// TIA Portal V15.1 export
// export: Created 2024-06-21T08:41:04.5665723Z, ExportSetting WithDefaults, DisplayName Totally Integrated Automation Portal, DisplayVersion V15.1 Update 5, DisplayName TIA Portal Openness, DisplayVersion V15.1 Update 5, DisplayName SINAMICS Startdrive Advanced, DisplayVersion V15.1, DisplayName G130, G150, S120, S150, SINAMICS MV, S210, DisplayVersion V15.1, DisplayName G110M, G120, G120C, G120D, G120P, DisplayVersion V15.1, DisplayName STEP 7 Professional, DisplayVersion V15.1 Update 5, DisplayName STEP 7 Safety, DisplayVersion V15.1, DisplayName WinCC Professional, DisplayVersion V15.1 Update 5, DisplayName SIMATIC Visualization Architect, DisplayVersion V15.1
FUNCTION_BLOCK "LProcVlvPidFbk"   // FB1734, FBD
TITLE = LProcVlvPidFbk
{ S7_Optimized_Access := 'FALSE' }
AUTHOR : VCC
FAMILY : ProcEq
NAME : PIDDONFb
VERSION : 0.1
// ================================================================================
// This is a Valve/Damper PID-controller module.
// The module contains: 
// 1 analog input function block
// a PID controller loop and a DO controller to activate the contactors Open
// and Close
// There is a feedback of position of the valve.
// ================================================================================
// stored: AutoNumber false, IsIECCheckEnabled false, SetENOAutomatically False, UDAEnableTagReadback false
   VAR_INPUT
      I_ExtSP1_Value { ExternalAccessible := 'False'; ExternalVisible := 'False'; ExternalWritable := 'False'} : Real;   // External Set-point 1
      I_ForcedValue { ExternalAccessible := 'False'; ExternalVisible := 'False'; ExternalWritable := 'False'} : Real;   // Pid Output Forced value (when I_ForceOutput is true)
      I_DO_POS { ExternalAccessible := 'False'; ExternalVisible := 'False'; ExternalWritable := 'False'} : Int;   // Feedback position DO controller
      I_DetSetLimit { ExternalAccessible := 'False'; ExternalVisible := 'False'; ExternalWritable := 'False'} : Real;   // Detection Set Limit
      I_DetResetLimit { ExternalAccessible := 'False'; ExternalVisible := 'False'; ExternalWritable := 'False'} : Real := 100.0;   // Detection Reset Limit
      I_PV_AnInput { ExternalAccessible := 'False'; ExternalVisible := 'False'; ExternalWritable := 'False'} : Int;   // Process Value Analog Input
      I_SPReq : Int;   // Index Set-point Request
      I_MaxTime { ExternalAccessible := 'False'; ExternalVisible := 'False'; ExternalWritable := 'False'} : DInt;   // Maximum Time to get Set and reset detections
      I_ExtSP1 { ExternalAccessible := 'False'; ExternalVisible := 'False'; ExternalWritable := 'False'} : Bool;   // External Set-point 1 Request
      I_ControllerON { ExternalAccessible := 'False'; ExternalVisible := 'False'; ExternalWritable := 'False'} : Bool;   // Start Pid Controller
      I_ForceOutput : Bool;   // Force Pid Output Value to Forced Value
      I_DetSet { ExternalAccessible := 'False'; ExternalVisible := 'False'; ExternalWritable := 'False'} : Bool;   // Detection Set
      I_DetReset { ExternalAccessible := 'False'; ExternalVisible := 'False'; ExternalWritable := 'False'} : Bool;   // Detection Reset
      I_AutoSetReq { ExternalAccessible := 'False'; ExternalVisible := 'False'; ExternalWritable := 'False'} : Bool;   // Set Valve/Damper from sequence or equation
      I_AutoResetReq { ExternalAccessible := 'False'; ExternalVisible := 'False'; ExternalWritable := 'False'} : Bool;   // Reset Valve/Damper from sequence or equation
      I_InterlockSetOk { ExternalAccessible := 'False'; ExternalVisible := 'False'; ExternalWritable := 'False'} : Bool;   // Interlock Set Direction
      I_InterlockResetOk { ExternalAccessible := 'False'; ExternalVisible := 'False'; ExternalWritable := 'False'} : Bool;   // Interlock Reset Direction
      I_EnableAlarm { ExternalAccessible := 'False'; ExternalVisible := 'False'; ExternalWritable := 'False'} : Bool;   // Enable Alarms
      I_PBSetPBResetAllAutoSel { ExternalAccessible := 'False'; ExternalVisible := 'False'; ExternalWritable := 'False'} : Struct   // Set PB activated - Reset PB activated - All HMI Auto selected
         HMI1SetPB { ExternalAccessible := 'False'; ExternalVisible := 'False'; ExternalWritable := 'False'} : Bool;   // Set PB activated on HMI1
         HMI1ResetPB { ExternalAccessible := 'False'; ExternalVisible := 'False'; ExternalWritable := 'False'} : Bool;   // Reset PB activated on HMI1
         HMI1AllHMIAutoSel { ExternalAccessible := 'False'; ExternalVisible := 'False'; ExternalWritable := 'False'} : Bool;   // All HMI Auto selected on HMI1
         HMI2SetPB { ExternalAccessible := 'False'; ExternalVisible := 'False'; ExternalWritable := 'False'} : Bool;   // Set PB activated on HMI2
         HMI2ResetPB { ExternalAccessible := 'False'; ExternalVisible := 'False'; ExternalWritable := 'False'} : Bool;   // Reset PB activated on HMI2
         HMI2AllHMIAutoSel { ExternalAccessible := 'False'; ExternalVisible := 'False'; ExternalWritable := 'False'} : Bool;   // All HMI Auto selected on HMI2
         HMI3SetPB { ExternalAccessible := 'False'; ExternalVisible := 'False'; ExternalWritable := 'False'} : Bool;   // Set PB activated on HMI3
         HMI3ResetPB { ExternalAccessible := 'False'; ExternalVisible := 'False'; ExternalWritable := 'False'} : Bool;   // Reset PB activated on HMI3
         HMI3AllHMIAutoSel { ExternalAccessible := 'False'; ExternalVisible := 'False'; ExternalWritable := 'False'} : Bool;   // All HMI Auto selected on HMI3
         HMI4SetPB { ExternalAccessible := 'False'; ExternalVisible := 'False'; ExternalWritable := 'False'} : Bool;   // Set PB activated on HMI4
         HMI4ResetPB { ExternalAccessible := 'False'; ExternalVisible := 'False'; ExternalWritable := 'False'} : Bool;   // Reset PB activated on HMI4
         HMI4AllHMIAutoSel { ExternalAccessible := 'False'; ExternalVisible := 'False'; ExternalWritable := 'False'} : Bool;   // All HMI Auto selected on HMI4
         HMI5SetPB { ExternalAccessible := 'False'; ExternalVisible := 'False'; ExternalWritable := 'False'} : Bool;   // Set PB activated on HMI5
         HMI5ResetPB { ExternalAccessible := 'False'; ExternalVisible := 'False'; ExternalWritable := 'False'} : Bool;   // Reset PB activated on HMI5
         HMI5AllHMIAutoSel { ExternalAccessible := 'False'; ExternalVisible := 'False'; ExternalWritable := 'False'} : Bool;   // All HMI Auto selected on HMI5
         StartPBSel { ExternalAccessible := 'False'; ExternalVisible := 'False'; ExternalWritable := 'False'} : Bool;   // Start is activated
         AlarmResetPBSel { ExternalAccessible := 'False'; ExternalVisible := 'False'; ExternalWritable := 'False'} : Bool;   // Alarm reset is activated
      END_STRUCT;
      I_UpperLevelAlarmA { ExternalAccessible := 'False'; ExternalVisible := 'False'; ExternalWritable := 'False'} : Bool;   // Alarm A from Upper Level
      I_UpperLevelAlarmB { ExternalAccessible := 'False'; ExternalVisible := 'False'; ExternalWritable := 'False'} : Bool;   // Alarm B from Upper Level
      I_EnHHHAlarm { ExternalAccessible := 'False'; ExternalVisible := 'False'; ExternalWritable := 'False'} : Bool;   // Enable HHH Limit Alarm
      I_ResHHHAlarm { ExternalAccessible := 'False'; ExternalVisible := 'False'; ExternalWritable := 'False'} : Bool;   // Reset HHH Limit Alarm
      I_EnHHAlarm { ExternalAccessible := 'False'; ExternalVisible := 'False'; ExternalWritable := 'False'} : Bool;   // Enable HH Limit Alarm
      I_ResHHAlarm { ExternalAccessible := 'False'; ExternalVisible := 'False'; ExternalWritable := 'False'} : Bool;   // Reset HH Limit Alarm
      I_EnHAlarm { ExternalAccessible := 'False'; ExternalVisible := 'False'; ExternalWritable := 'False'} : Bool;   // Enable H Limit Alarm
      I_ResHAlarm { ExternalAccessible := 'False'; ExternalVisible := 'False'; ExternalWritable := 'False'} : Bool;   // Reset H Limit Alarm
      I_EnLAlarm { ExternalAccessible := 'False'; ExternalVisible := 'False'; ExternalWritable := 'False'} : Bool;   // Enable L Limit Alarm
      I_ResLAlarm { ExternalAccessible := 'False'; ExternalVisible := 'False'; ExternalWritable := 'False'} : Bool;   // Reset L Limit Alarm
      I_EnLLAlarm { ExternalAccessible := 'False'; ExternalVisible := 'False'; ExternalWritable := 'False'} : Bool;   // Enable LL Limit Alarm
      I_ResLLAlarm { ExternalAccessible := 'False'; ExternalVisible := 'False'; ExternalWritable := 'False'} : Bool;   // Reset LL Limit Alarm
      I_EnLLLAlarm { ExternalAccessible := 'False'; ExternalVisible := 'False'; ExternalWritable := 'False'} : Bool;   // Enable LLL Limit Alarm
      I_ResLLLAlarm { ExternalAccessible := 'False'; ExternalVisible := 'False'; ExternalWritable := 'False'} : Bool;   // Reset LLL Limit Alarm
      C_ManualForcedUsed { ExternalAccessible := 'False'; ExternalVisible := 'False'; ExternalWritable := 'False'} : Bool;   // Manual Forced is used (=true)
      C_DetSetUsed { ExternalAccessible := 'False'; ExternalVisible := 'False'; ExternalWritable := 'False'} : Bool;   // Detection Set used (true=used)
      C_DetResetUsed { ExternalAccessible := 'False'; ExternalVisible := 'False'; ExternalWritable := 'False'} : Bool;   // Detection Reset used (true=used)
   END_VAR
   VAR_OUTPUT
      O_PV : Real;   // Process Value scaled
      O_SP : Real;   // Setpoint used in controller
      O_PosFbk : Real;   // Damp/Valve position feedback value used in controller
      O_LMN : Real;   // Pid Output value
      O_SetFbk : Bool;   // Valve/Damper in Set position
      O_ResetFbk : Bool;   // Valve/Damper in Reset position
      O_SetCmd { ExternalAccessible := 'False'; ExternalVisible := 'False'; ExternalWritable := 'False'} : Bool;   // Valve/Damper Set command
      O_ResetCmd { ExternalAccessible := 'False'; ExternalVisible := 'False'; ExternalWritable := 'False'} : Bool;   // Valve/Damper Reset command
      O_AlarmABCondition { ExternalAccessible := 'False'; ExternalVisible := 'False'; ExternalWritable := 'False'} : Bool;   // Alarm AB condition
      O_AlarmA { ExternalAccessible := 'False'; ExternalVisible := 'False'; ExternalWritable := 'False'} : Bool;   // Summation Alarm A
      O_AlarmB { ExternalAccessible := 'False'; ExternalVisible := 'False'; ExternalWritable := 'False'} : Bool;   // Summation Alarm B
      O_AlarmC { ExternalAccessible := 'False'; ExternalVisible := 'False'; ExternalWritable := 'False'} : Bool;   // Summation Alarm C
      O_AlarmD { ExternalAccessible := 'False'; ExternalVisible := 'False'; ExternalWritable := 'False'} : Bool;   // Summation Alarm D
      O_HHHAlarm { ExternalAccessible := 'False'; ExternalVisible := 'False'; ExternalWritable := 'False'} : Bool;   // HHH Alarm
      O_HHAlarm { ExternalAccessible := 'False'; ExternalVisible := 'False'; ExternalWritable := 'False'} : Bool;   // HH Alarm
      O_HAlarm { ExternalAccessible := 'False'; ExternalVisible := 'False'; ExternalWritable := 'False'} : Bool;   // H Alarm
      O_LAlarm { ExternalAccessible := 'False'; ExternalVisible := 'False'; ExternalWritable := 'False'} : Bool;   // L Alarm
      O_LLAlarm { ExternalAccessible := 'False'; ExternalVisible := 'False'; ExternalWritable := 'False'} : Bool;   // LL Alarm
      O_LLLAlarm { ExternalAccessible := 'False'; ExternalVisible := 'False'; ExternalWritable := 'False'} : Bool;   // LLL Alarm
      O_HHHReached { ExternalAccessible := 'False'; ExternalVisible := 'False'; ExternalWritable := 'False'} : Bool;   // High High High Limit Reached
      O_HHReached { ExternalAccessible := 'False'; ExternalVisible := 'False'; ExternalWritable := 'False'} : Bool;   // High High Limit Reached
      O_HReached { ExternalAccessible := 'False'; ExternalVisible := 'False'; ExternalWritable := 'False'} : Bool;   // High Limit Reached
      O_LReached { ExternalAccessible := 'False'; ExternalVisible := 'False'; ExternalWritable := 'False'} : Bool;   // Low Limit Reached
      O_LLReached { ExternalAccessible := 'False'; ExternalVisible := 'False'; ExternalWritable := 'False'} : Bool;   // Low Low Limit Reached
      O_LLLReached { ExternalAccessible := 'False'; ExternalVisible := 'False'; ExternalWritable := 'False'} : Bool;   // Low Low Low Limit Reached
      H_IAnim { ExternalAccessible := 'False'; ExternalVisible := 'False'; ExternalWritable := 'False'} : Word;   // HMI Animation color of the icon
      H_AlarmWord { ExternalAccessible := 'False'; ExternalVisible := 'False'; ExternalWritable := 'False'} : DWord;   // Alarm Word
   END_VAR
   VAR_IN_OUT
      PV_AnScale : "LProcAnInput6Lim";   // DB for the analogue scaling of Process Value
   END_VAR
   VAR DB_SPECIFIC
      AB_OvTimeAutoSel { ExternalAccessible := 'False'; ExternalVisible := 'False'; ExternalWritable := 'False'} : Bool;   // Alarm Overtime Auto selected
      AD_AcofDetSet { ExternalAccessible := 'False'; ExternalVisible := 'False'; ExternalWritable := 'False'} : Bool;   // Acof Fault Set detection
      AD_AcofDetReset { ExternalAccessible := 'False'; ExternalVisible := 'False'; ExternalWritable := 'False'} : Bool;   // Acof Fault Reset detection
      AD_PV_SensorAlm { ExternalAccessible := 'False'; ExternalVisible := 'False'; ExternalWritable := 'False'} : Bool;   // Process Value sensor alarm
      AD_InterlockSetAlm { ExternalAccessible := 'False'; ExternalVisible := 'False'; ExternalWritable := 'False'} : Bool;   // Interlock Set Alarm
      AD_InterlockResetAlm { ExternalAccessible := 'False'; ExternalVisible := 'False'; ExternalWritable := 'False'} : Bool;   // Interlock Reset Alarm
      H_HMIModeCmd : Word;   // Mode commands from HMI
      H_ActiveHMI : Int;   // Active HMI
      H_NameActiveHMI : String[25];   // Name of the Active HMI
      H_In : Struct   // HMI
         SP2 : Real;   // Set-point 2
         SP3 : Real;   // Set-point 3
         SP4 : Real;   // Set-point 4
         SP5 : Real;   // Set-point 5
         GAIN : Real;   // Pid Proportional Gain
         PID_DEADB_W : Real;   // Pid Deadband width
         LMN_HLM : Real;   // Pid Manipulated value high limit
         LMN_LLM : Real;   // Pid Manipulated value low limit
         TI : Time;   // Pid Reset time
         TD : Time;   // Pid Derivative time
         PULSE_TM : Time;   // Minimum Pulse Time
         BREAK_TM : Time;   // Minimum Break Time
         MTR_TM : Time;   // Motor manipulated time value
         DO_DEADB_W : Real;   // Motor Deadband width
         DO_POS_FAC : Real;   // Factor for feedback of position
         Direct : Bool;   // Pid in Direct mode (output increase if SP>PV)
         P_SEL : Bool;   // Pid P selected
         I_SEL : Bool;   // Pid I selected
         D_SEL : Bool;   // Pid D selected
      END_STRUCT;
      H_Out : Struct   // HMI
         AnInputIAnim : Word;   // HMI Animation color of the icon
         DetSetIAnim : Word;   // HMI Animation color of object
         DetResetIAnim : Word;   // HMI Animation color of object
         ContactorSetIAnim : Word;   // HMI Animation color of object
         ContactorResetIAnim : Word;   // HMI Animation color of object
         Anim : Word;   // HMI Animation of the object
         Anim2 : Word;   // HMI Animation of the object
         Anim3 : Bool;   // HMI Animation bool
         DBnr : Int;   // HMI Animation DB number
      END_STRUCT;
      H_InOut : Struct   // HMI
         Manual_Value : Real;   // Position Setpoint in Manual
         SP1 : Real;   // Set-point 1
      END_STRUCT;
      CYCLE { ExternalAccessible := 'False'; ExternalVisible := 'False'; ExternalWritable := 'False'} : Time := T#100MS;   // Sample time for controller
      PV_AIScaled { ExternalAccessible := 'False'; ExternalVisible := 'False'; ExternalWritable := 'False'} : Real;   // Proces Value: Analog Input after scaling
      PV_PID { ExternalAccessible := 'False'; ExternalVisible := 'False'; ExternalWritable := 'False'} : Real;   // Pid Process value
      SPSel { ExternalAccessible := 'False'; ExternalVisible := 'False'; ExternalWritable := 'False'} : Real;   // Set-point selected
      SP { ExternalAccessible := 'False'; ExternalVisible := 'False'; ExternalWritable := 'False'} : Real;   // Set-point used for Pid regulation
      PosFbk { ExternalAccessible := 'False'; ExternalVisible := 'False'; ExternalWritable := 'False'} : Real;   // Position Feedback (calculation) of the Valve/Damper
      DeadPosOpen { ExternalAccessible := 'False'; ExternalVisible := 'False'; ExternalWritable := 'False'} : Real;   // Calculation Position Open - deadband
      DeadPosClosed { ExternalAccessible := 'False'; ExternalVisible := 'False'; ExternalWritable := 'False'} : Real;   // Calculation Position Closed + deadband
      LMN { ExternalAccessible := 'False'; ExternalVisible := 'False'; ExternalWritable := 'False'} : Real;   // Pid Output value
      DetSet { ExternalAccessible := 'False'; ExternalVisible := 'False'; ExternalWritable := 'False'} : Bool;   // Detection Set
      DetReset { ExternalAccessible := 'False'; ExternalVisible := 'False'; ExternalWritable := 'False'} : Bool;   // Detection Reset
      AutoMode { ExternalAccessible := 'False'; ExternalVisible := 'False'; ExternalWritable := 'False'} : Bool;   // Auto mode
      ManualMode { ExternalAccessible := 'False'; ExternalVisible := 'False'; ExternalWritable := 'False'} : Bool;   // Manual mode
      AutoModeSel { ExternalAccessible := 'False'; ExternalVisible := 'False'; ExternalWritable := 'False'} : Bool;   // Auto Mode Selection from HMI
      ManualModeSel { ExternalAccessible := 'False'; ExternalVisible := 'False'; ExternalWritable := 'False'} : Bool;   // Manual Mode Selection from HMI
      ForcedMan { ExternalAccessible := 'False'; ExternalVisible := 'False'; ExternalWritable := 'False'} : Bool;   // Forced manual active
      AllHMIAutoSel { ExternalAccessible := 'False'; ExternalVisible := 'False'; ExternalWritable := 'False'} : Bool;   // All HMI Auto selected
      Set { ExternalAccessible := 'False'; ExternalVisible := 'False'; ExternalWritable := 'False'} : Bool;   // Controller output Set
      Reset { ExternalAccessible := 'False'; ExternalVisible := 'False'; ExternalWritable := 'False'} : Bool;   // Controller output Reset
      OvTimeAutoSelCond { ExternalAccessible := 'False'; ExternalVisible := 'False'; ExternalWritable := 'False'} : Bool;   // Overtime Auto selected condition
      SetCmd { ExternalAccessible := 'False'; ExternalVisible := 'False'; ExternalWritable := 'False'} : Bool;   // Set Command Request after interlock
      ResetCmd { ExternalAccessible := 'False'; ExternalVisible := 'False'; ExternalWritable := 'False'} : Bool;   // Reset Command Request after interlock
      Active { ExternalAccessible := 'False'; ExternalVisible := 'False'; ExternalWritable := 'False'} : Bool;   // Valve/Damper loop active
      AlarmA { ExternalAccessible := 'False'; ExternalVisible := 'False'; ExternalWritable := 'False'} : Bool;   // Summation Alarm A
      AlarmB { ExternalAccessible := 'False'; ExternalVisible := 'False'; ExternalWritable := 'False'} : Bool;   // Summation Alarm B
      AlarmC { ExternalAccessible := 'False'; ExternalVisible := 'False'; ExternalWritable := 'False'} : Bool;   // Summation Alarm C
      AlarmD { ExternalAccessible := 'False'; ExternalVisible := 'False'; ExternalWritable := 'False'} : Bool;   // Summation Alarm D
      DBnr { ExternalAccessible := 'False'; ExternalVisible := 'False'; ExternalWritable := 'False'} : Int;   // HMI DB number
   END_VAR
   VAR
      DetectionSet { ExternalAccessible := 'False'; ExternalVisible := 'False'; ExternalWritable := 'False'; S7_SetPoint := 'True'} : "LProcAcofDet";   // Detection SET
      DetectionReset { ExternalAccessible := 'False'; ExternalVisible := 'False'; ExternalWritable := 'False'; S7_SetPoint := 'True'} : "LProcAcofDet";   // Detection RESET
      PIDSelSP { ExternalAccessible := 'False'; ExternalVisible := 'False'; ExternalWritable := 'False'; S7_SetPoint := 'True'} : "LProcSel5SP";   // PID SP-selection between 5 Setpoint
      PID { ExternalAccessible := 'False'; ExternalVisible := 'False'; ExternalWritable := 'False'; S7_SetPoint := 'True'} : "LProcPid";   // PID Controller settings
      I_DO { ExternalAccessible := 'False'; ExternalVisible := 'False'; ExternalWritable := 'False'; S7_SetPoint := 'True'} : "LProcDO_Fbk";   // PID Converter to Digital
      Modes { ExternalAccessible := 'False'; ExternalVisible := 'False'; ExternalWritable := 'False'; S7_SetPoint := 'True'} : "LProcObjectMode";
   END_VAR
   VAR DB_SPECIFIC
      CheckActiveHMI { ExternalAccessible := 'False'; ExternalVisible := 'False'; ExternalWritable := 'False'; S7_SetPoint := 'True'} : TP_TIME;   // Timer
      CheckActiveHMI_1 { ExternalAccessible := 'False'; ExternalVisible := 'False'; ExternalWritable := 'False'; S7_SetPoint := 'True'} : TP_TIME;   // Timer
      CheckActiveHMI_2 { ExternalAccessible := 'False'; ExternalVisible := 'False'; ExternalWritable := 'False'; S7_SetPoint := 'True'} : TON_TIME;   // Timer
      CheckActiveHMI_3 { ExternalAccessible := 'False'; ExternalVisible := 'False'; ExternalWritable := 'False'; S7_SetPoint := 'True'} : TON_TIME;   // Timer
   END_VAR
   VAR_TEMP
      __PlcmigTempFillBits_0B0 : Array[0..15] of Bool;
   END_VAR
BEGIN

NETWORK
TITLE = **** 1 - Inputs **** DB number
// DB number
      L     DINO;
      T     #DBnr;

REGION Network 2: **** 1 - Inputs **** Temperature channel 1: Scaling
   // Temperature channel 1: Scaling
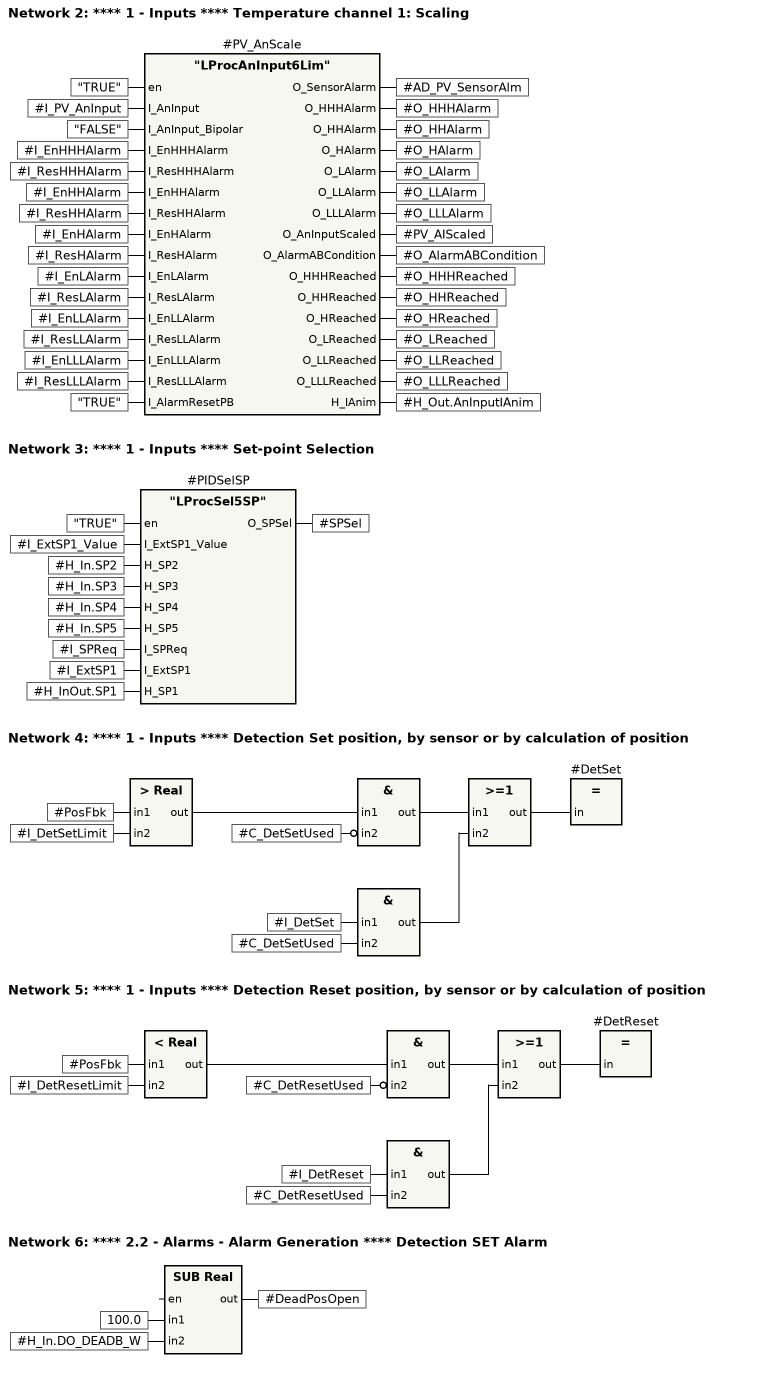
   IF "TRUE" THEN
       #PV_AnScale(I_AnInput := #I_PV_AnInput,   // "LProcAnInput6Lim"
                   I_AnInput_Bipolar := "FALSE",
                   I_EnHHHAlarm := #I_EnHHHAlarm,
                   I_ResHHHAlarm := #I_ResHHHAlarm,
                   I_EnHHAlarm := #I_EnHHAlarm,
                   I_ResHHAlarm := #I_ResHHAlarm,
                   I_EnHAlarm := #I_EnHAlarm,
                   I_ResHAlarm := #I_ResHAlarm,
                   I_EnLAlarm := #I_EnLAlarm,
                   I_ResLAlarm := #I_ResLAlarm,
                   I_EnLLAlarm := #I_EnLLAlarm,
                   I_ResLLAlarm := #I_ResLLAlarm,
                   I_EnLLLAlarm := #I_EnLLLAlarm,
                   I_ResLLLAlarm := #I_ResLLLAlarm,
                   I_AlarmResetPB := "TRUE",
                   O_SensorAlarm => #AD_PV_SensorAlm,
                   O_HHHAlarm => #O_HHHAlarm,
                   O_HHAlarm => #O_HHAlarm,
                   O_HAlarm => #O_HAlarm,
                   O_LAlarm => #O_LAlarm,
                   O_LLAlarm => #O_LLAlarm,
                   O_LLLAlarm => #O_LLLAlarm,
                   O_AnInputScaled => #PV_AIScaled,
                   O_AlarmABCondition => #O_AlarmABCondition,
                   O_HHHReached => #O_HHHReached,
                   O_HHReached => #O_HHReached,
                   O_HReached => #O_HReached,
                   O_LReached => #O_LReached,
                   O_LLReached => #O_LLReached,
                   O_LLLReached => #O_LLLReached,
                   H_IAnim => #H_Out.AnInputIAnim);
   END_IF;
END_REGION

REGION Network 3: **** 1 - Inputs **** Set-point Selection
   // Set-point Selection
   IF "TRUE" THEN
       #PIDSelSP(I_ExtSP1_Value := #I_ExtSP1_Value,   // "LProcSel5SP"
                 H_SP2 := #H_In.SP2,
                 H_SP3 := #H_In.SP3,
                 H_SP4 := #H_In.SP4,
                 H_SP5 := #H_In.SP5,
                 I_SPReq := #I_SPReq,
                 I_ExtSP1 := #I_ExtSP1,
                 H_SP1 := #H_InOut.SP1,
                 O_SPSel => #SPSel);
   END_IF;
END_REGION

REGION Network 4: **** 1 - Inputs **** Detection Set position, by sensor or by calculation of position
   // Detection Set position, by sensor or by calculation of position
   #DetSet := ((#PosFbk > #I_DetSetLimit) AND NOT #C_DetSetUsed) OR (#I_DetSet AND #C_DetSetUsed);
END_REGION

REGION Network 5: **** 1 - Inputs **** Detection Reset position, by sensor or by calculation of position
   // Detection Reset position, by sensor or by calculation of position
   #DetReset := ((#PosFbk < #I_DetResetLimit) AND NOT #C_DetResetUsed) OR (#I_DetReset AND #C_DetResetUsed);
END_REGION

REGION Network 6: **** 2.2 - Alarms - Alarm Generation **** Detection SET Alarm
   // Calculation Position Open - deadband
   #DeadPosOpen := 100.0 - #H_In.DO_DEADB_W;
END_REGION

REGION Network 7: **** 2.2 - Alarms - Alarm Generation **** Detection SET Alarm
   // Detection SET Alarm
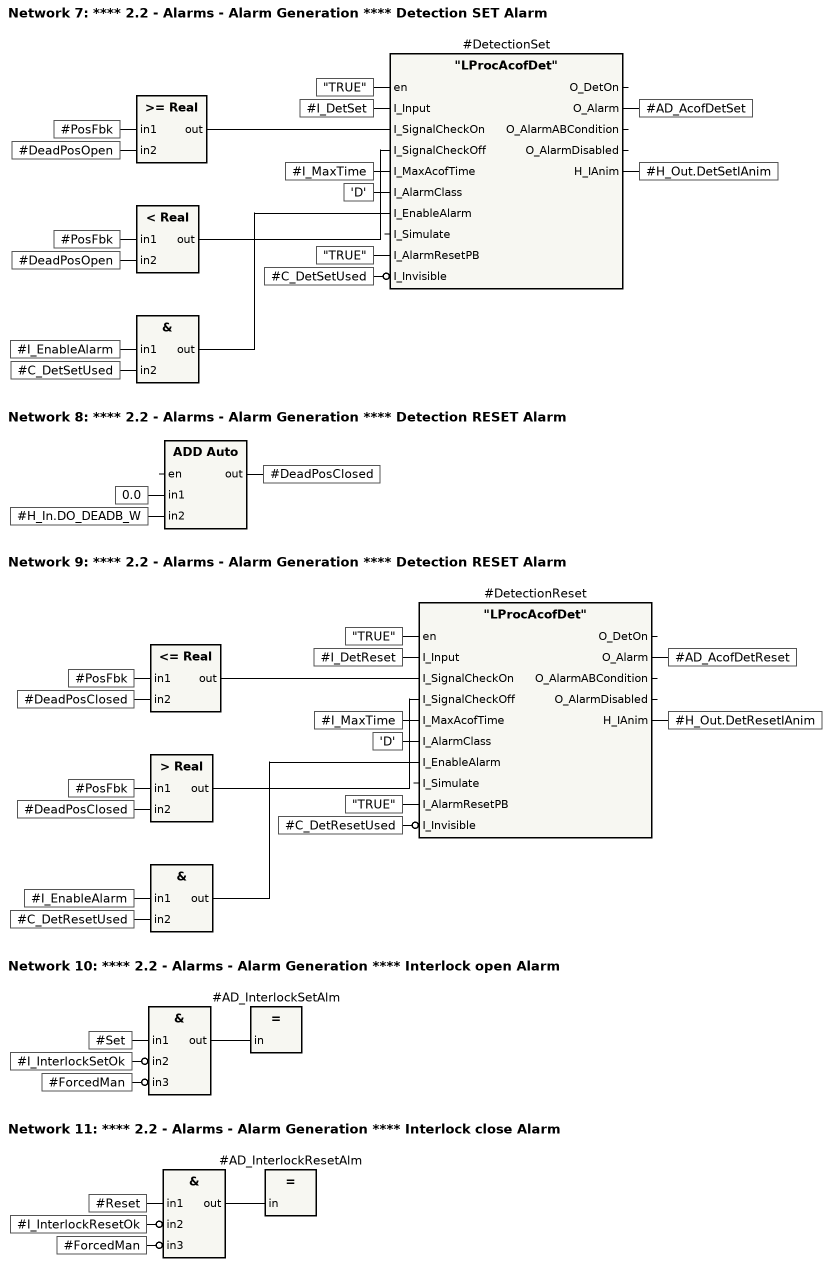
   IF "TRUE" THEN
       #DetectionSet(I_Input := #I_DetSet,   // "LProcAcofDet"
                     I_SignalCheckOn := #PosFbk >= #DeadPosOpen,
                     I_SignalCheckOff := #PosFbk < #DeadPosOpen,
                     I_MaxAcofTime := #I_MaxTime,
                     I_AlarmClass := 'D',
                     I_EnableAlarm := #I_EnableAlarm AND #C_DetSetUsed,
                     I_AlarmResetPB := "TRUE",
                     I_Invisible := NOT #C_DetSetUsed,
                     O_Alarm => #AD_AcofDetSet,
                     H_IAnim => #H_Out.DetSetIAnim);
   END_IF;
END_REGION

REGION Network 8: **** 2.2 - Alarms - Alarm Generation **** Detection RESET Alarm
   // Calculation Position Closed + deadband
   #DeadPosClosed := 0.0 + #H_In.DO_DEADB_W;
END_REGION

REGION Network 9: **** 2.2 - Alarms - Alarm Generation **** Detection RESET Alarm
   // Detection RESET Alarm
   IF "TRUE" THEN
       #DetectionReset(I_Input := #I_DetReset,   // "LProcAcofDet"
                       I_SignalCheckOn := #PosFbk <= #DeadPosClosed,
                       I_SignalCheckOff := #PosFbk > #DeadPosClosed,
                       I_MaxAcofTime := #I_MaxTime,
                       I_AlarmClass := 'D',
                       I_EnableAlarm := #I_EnableAlarm AND #C_DetResetUsed,
                       I_AlarmResetPB := "TRUE",
                       I_Invisible := NOT #C_DetResetUsed,
                       O_Alarm => #AD_AcofDetReset,
                       H_IAnim => #H_Out.DetResetIAnim);
   END_IF;
END_REGION

REGION Network 10: **** 2.2 - Alarms - Alarm Generation **** Interlock open Alarm
   // Interlock open Alarm
   #AD_InterlockSetAlm := #Set AND NOT #I_InterlockSetOk AND NOT #ForcedMan;
END_REGION

REGION Network 11: **** 2.2 - Alarms - Alarm Generation **** Interlock close Alarm
   // Interlock close Alarm
   #AD_InterlockResetAlm := #Reset AND NOT #I_InterlockResetOk AND NOT #ForcedMan;
END_REGION

REGION Network 12: **** 4.5 - Machine Status - Modes **** Modes
   // Modes
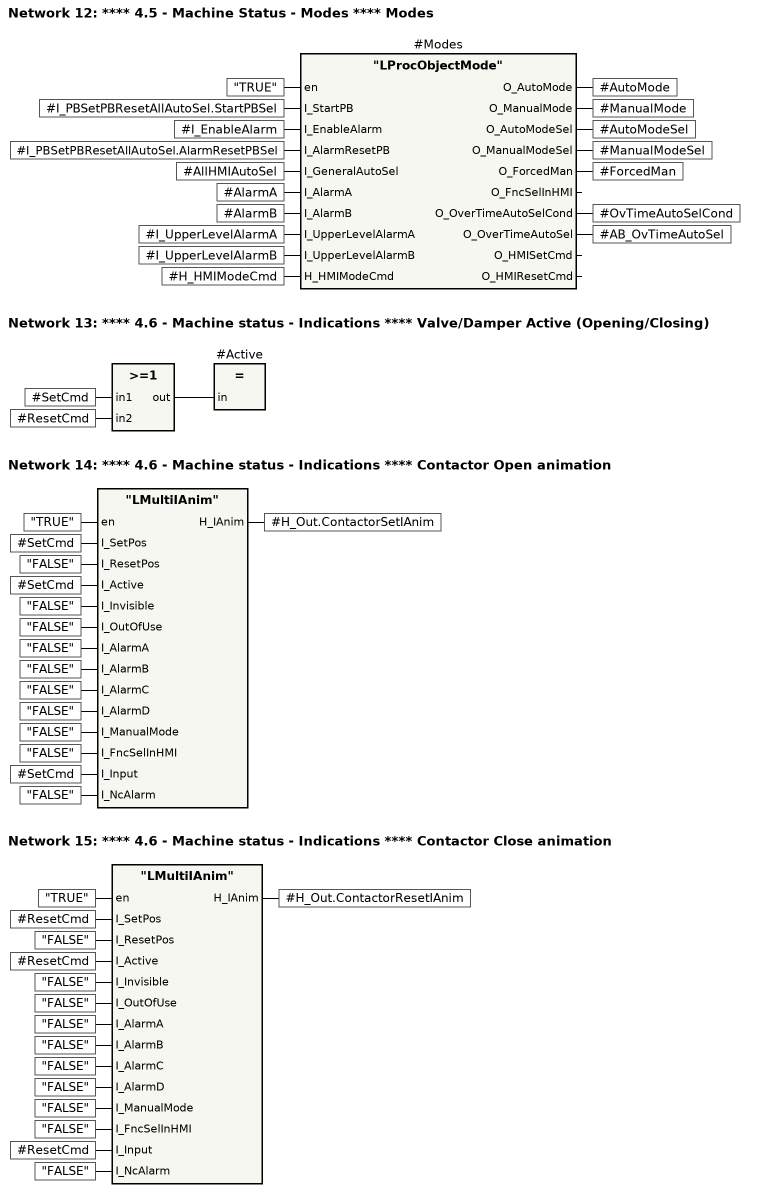
   IF "TRUE" THEN
       #Modes(I_StartPB := #I_PBSetPBResetAllAutoSel.StartPBSel,   // "LProcObjectMode"
              I_EnableAlarm := #I_EnableAlarm,
              I_AlarmResetPB := #I_PBSetPBResetAllAutoSel.AlarmResetPBSel,
              I_GeneralAutoSel := #AllHMIAutoSel,
              I_AlarmA := #AlarmA,
              I_AlarmB := #AlarmB,
              I_UpperLevelAlarmA := #I_UpperLevelAlarmA,
              I_UpperLevelAlarmB := #I_UpperLevelAlarmB,
              H_HMIModeCmd := #H_HMIModeCmd,
              O_AutoMode => #AutoMode,
              O_ManualMode => #ManualMode,
              O_AutoModeSel => #AutoModeSel,
              O_ManualModeSel => #ManualModeSel,
              O_ForcedMan => #ForcedMan,
              O_OverTimeAutoSelCond => #OvTimeAutoSelCond,
              O_OverTimeAutoSel => #AB_OvTimeAutoSel);
   END_IF;
END_REGION

REGION Network 13: **** 4.6 - Machine status - Indications **** Valve/Damper Active (Opening/Closing)
   // Valve/Damper Active (Opening/Closing)
   #Active := #SetCmd OR #ResetCmd;
END_REGION

REGION Network 14: **** 4.6 - Machine status - Indications **** Contactor Open animation
   // Contactor Open animation
   IF "TRUE" THEN
       "LMultiIAnim"(I_SetPos := #SetCmd,
                     I_ResetPos := "FALSE",
                     I_Active := #SetCmd,
                     I_Invisible := "FALSE",
                     I_OutOfUse := "FALSE",
                     I_AlarmA := "FALSE",
                     I_AlarmB := "FALSE",
                     I_AlarmC := "FALSE",
                     I_AlarmD := "FALSE",
                     I_ManualMode := "FALSE",
                     I_FncSelInHMI := "FALSE",
                     I_Input := #SetCmd,
                     I_NcAlarm := "FALSE",
                     H_IAnim => #H_Out.ContactorSetIAnim);
   END_IF;
END_REGION

REGION Network 15: **** 4.6 - Machine status - Indications **** Contactor Close animation
   // Contactor Close animation
   IF "TRUE" THEN
       "LMultiIAnim"(I_SetPos := #ResetCmd,
                     I_ResetPos := "FALSE",
                     I_Active := #ResetCmd,
                     I_Invisible := "FALSE",
                     I_OutOfUse := "FALSE",
                     I_AlarmA := "FALSE",
                     I_AlarmB := "FALSE",
                     I_AlarmC := "FALSE",
                     I_AlarmD := "FALSE",
                     I_ManualMode := "FALSE",
                     I_FncSelInHMI := "FALSE",
                     I_Input := #ResetCmd,
                     I_NcAlarm := "FALSE",
                     H_IAnim => #H_Out.ContactorResetIAnim);
   END_IF;
END_REGION

REGION Network 16: **** 4.6 - Machine status - Indications **** Icon animation
   // Icon animation
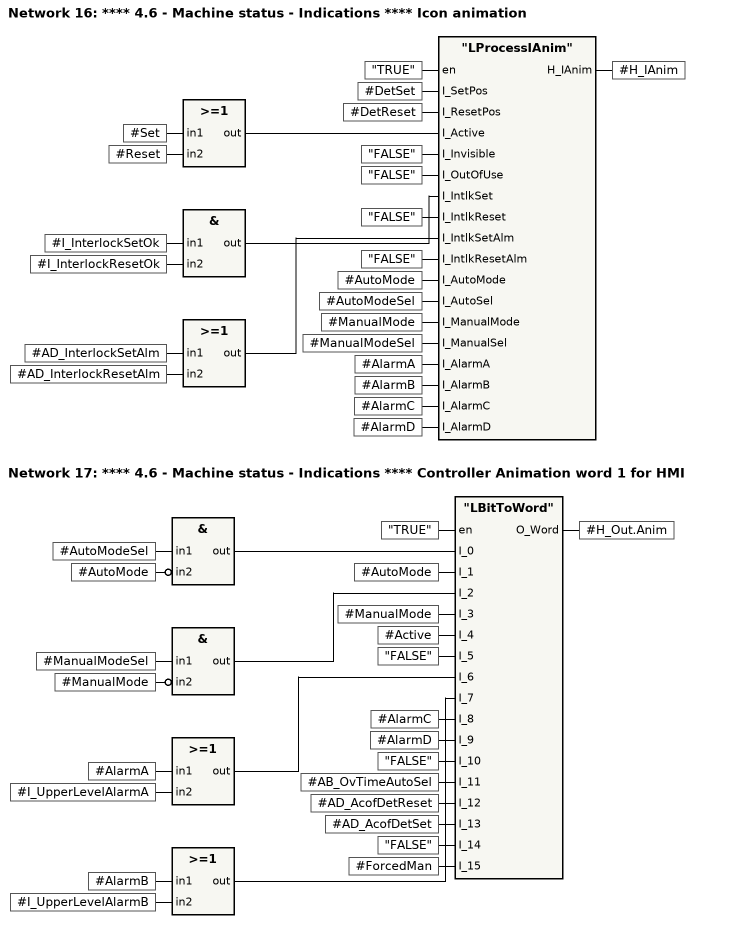
   IF "TRUE" THEN
       "LProcessIAnim"(I_SetPos := #DetSet,
                       I_ResetPos := #DetReset,
                       I_Active := #Set OR #Reset,
                       I_Invisible := "FALSE",
                       I_OutOfUse := "FALSE",
                       I_IntlkSet := #I_InterlockSetOk AND #I_InterlockResetOk,
                       I_IntlkReset := "FALSE",
                       I_IntlkSetAlm := #AD_InterlockSetAlm OR #AD_InterlockResetAlm,
                       I_IntlkResetAlm := "FALSE",
                       I_AutoMode := #AutoMode,
                       I_AutoSel := #AutoModeSel,
                       I_ManualMode := #ManualMode,
                       I_ManualSel := #ManualModeSel,
                       I_AlarmA := #AlarmA,
                       I_AlarmB := #AlarmB,
                       I_AlarmC := #AlarmC,
                       I_AlarmD := #AlarmD,
                       H_IAnim => #H_IAnim);
   END_IF;
END_REGION

REGION Network 17: **** 4.6 - Machine status - Indications **** Controller Animation word 1 for HMI
   // Controller Animation word 1 for HMI
   IF "TRUE" THEN
       "LBitToWord"(I_0 := #AutoModeSel AND NOT #AutoMode,
                    I_1 := #AutoMode,
                    I_2 := #ManualModeSel AND NOT #ManualMode,
                    I_3 := #ManualMode,
                    I_4 := #Active,
                    I_5 := "FALSE",
                    I_6 := #AlarmA OR #I_UpperLevelAlarmA,
                    I_7 := #AlarmB OR #I_UpperLevelAlarmB,
                    I_8 := #AlarmC,
                    I_9 := #AlarmD,
                    I_10 := "FALSE",
                    I_11 := #AB_OvTimeAutoSel,
                    I_12 := #AD_AcofDetReset,
                    I_13 := #AD_AcofDetSet,
                    I_14 := "FALSE",
                    I_15 := #ForcedMan,
                    O_Word => #H_Out.Anim);
   END_IF;
END_REGION

REGION Network 18: **** 4.6 - Machine status - Indications **** Controller Animation word 2 for HMI
   // Controller Animation word 2 for HMI
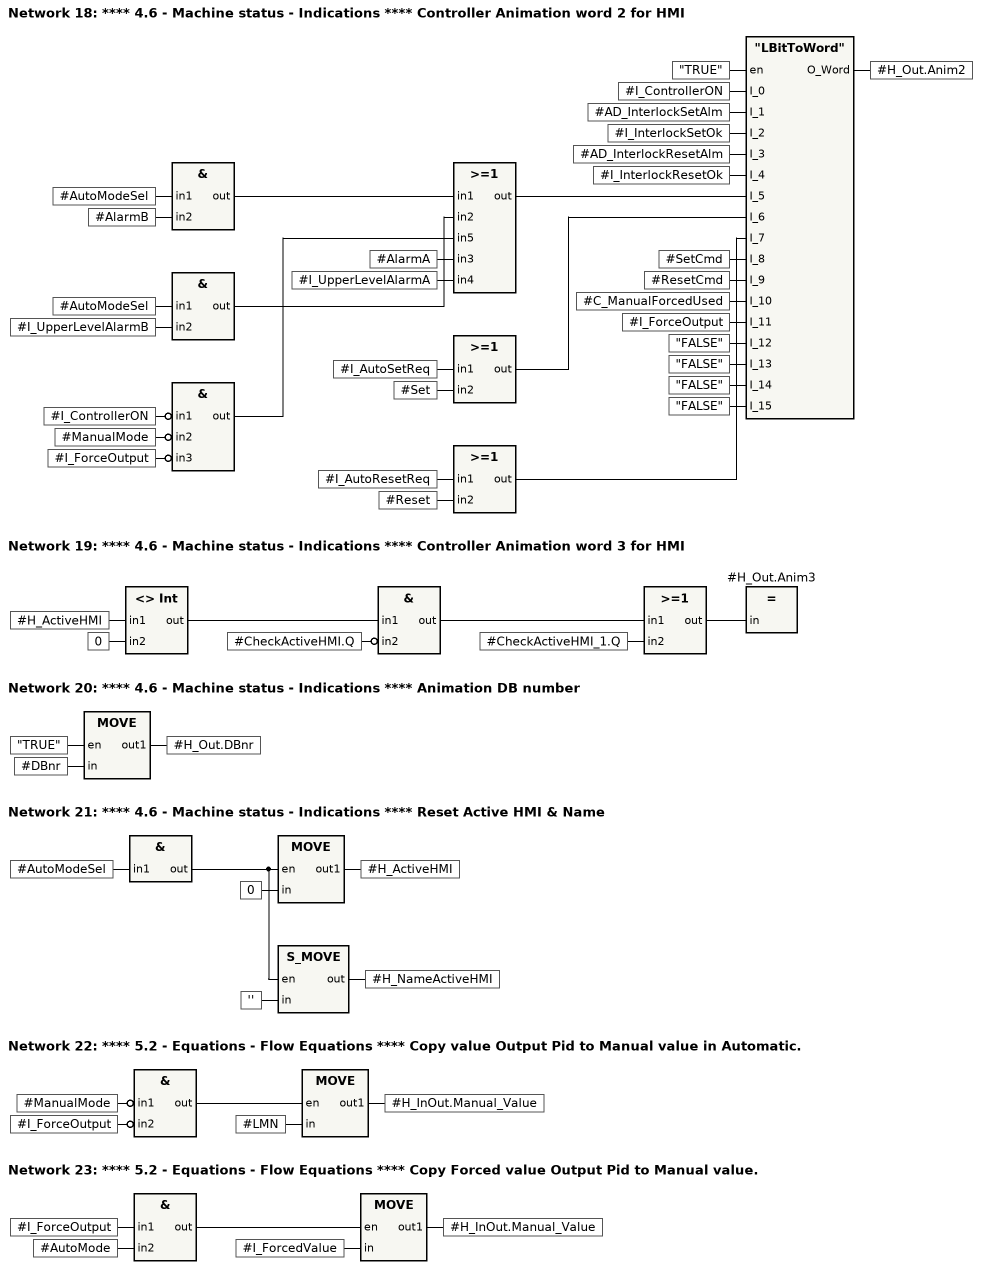
   IF "TRUE" THEN
       "LBitToWord"(I_0 := #I_ControllerON,
                    I_1 := #AD_InterlockSetAlm,
                    I_2 := #I_InterlockSetOk,
                    I_3 := #AD_InterlockResetAlm,
                    I_4 := #I_InterlockResetOk,
                    I_5 := (#AutoModeSel AND #AlarmB) OR (#AutoModeSel AND #I_UpperLevelAlarmB) OR (NOT #I_ControllerON AND NOT #ManualMode AND NOT #I_ForceOutput) OR #AlarmA OR #I_UpperLevelAlarmA,
                    I_6 := #I_AutoSetReq OR #Set,
                    I_7 := #I_AutoResetReq OR #Reset,
                    I_8 := #SetCmd,
                    I_9 := #ResetCmd,
                    I_10 := #C_ManualForcedUsed,
                    I_11 := #I_ForceOutput,
                    I_12 := "FALSE",
                    I_13 := "FALSE",
                    I_14 := "FALSE",
                    I_15 := "FALSE",
                    O_Word => #H_Out.Anim2);
   END_IF;
END_REGION

REGION Network 19: **** 4.6 - Machine status - Indications **** Controller Animation word 3 for HMI
   // Controller Animation word 3 for HMI
   #H_Out.Anim3 := ((#H_ActiveHMI <> 0) AND NOT #CheckActiveHMI.Q) OR #CheckActiveHMI_1.Q;
END_REGION

REGION Network 20: **** 4.6 - Machine status - Indications **** Animation DB number
   // Animation DB number
   IF "TRUE" THEN #H_Out.DBnr := #DBnr; END_IF;
END_REGION

REGION Network 21: **** 4.6 - Machine status - Indications **** Reset Active HMI & Name
   // Reset Active HMI & Name
   IF #AutoModeSel THEN
       #H_ActiveHMI := 0;
       #H_NameActiveHMI := '';
   END_IF;
END_REGION

REGION Network 22: **** 5.2 - Equations - Flow Equations **** Copy value Output Pid to Manual value in Automatic.
   // Copy value Output Pid to Manual value in Automatic.
   IF NOT #ManualMode AND NOT #I_ForceOutput THEN #H_InOut.Manual_Value := #LMN; END_IF;
END_REGION

REGION Network 23: **** 5.2 - Equations - Flow Equations **** Copy Forced value Output Pid to Manual value.
   // Copy Forced value Output Pid to Manual value.
   IF #I_ForceOutput AND #AutoMode THEN #H_InOut.Manual_Value := #I_ForcedValue; END_IF;
END_REGION

REGION Network 24: **** 5.2 - Equations - Flow **** All HMI Auto selected
   // All HMI Auto selected
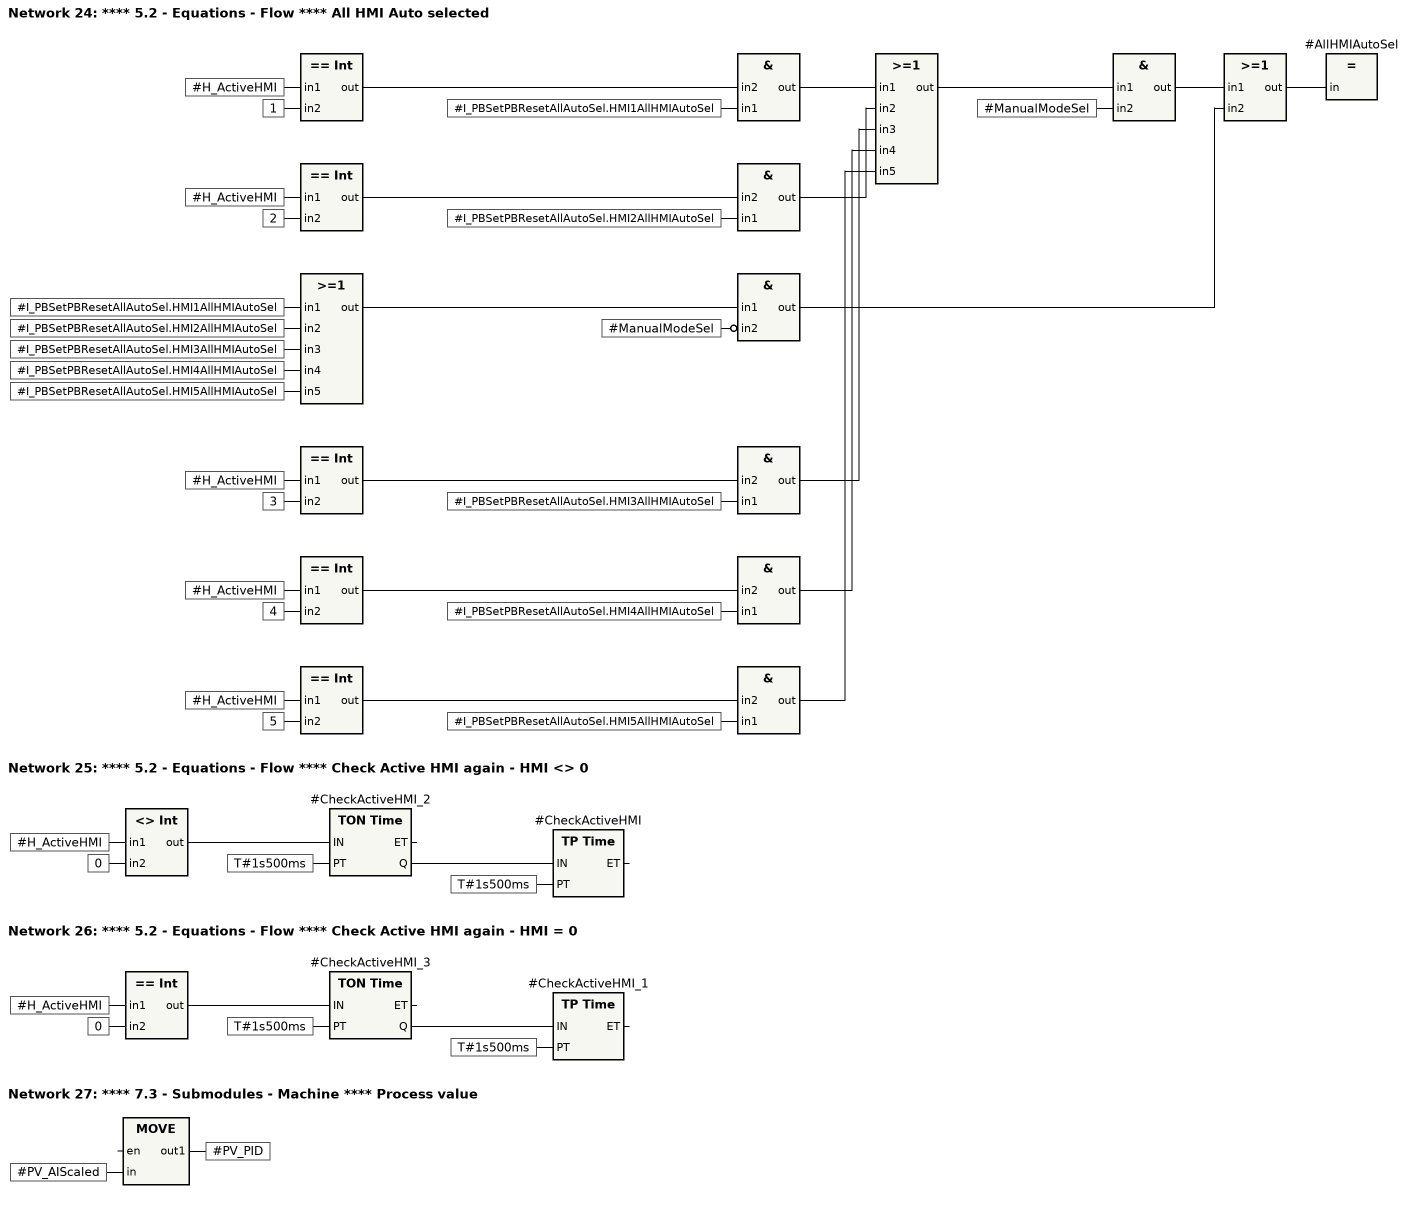
   #AllHMIAutoSel := ((((#H_ActiveHMI = 1) AND #I_PBSetPBResetAllAutoSel.HMI1AllHMIAutoSel) OR ((#H_ActiveHMI = 2) AND #I_PBSetPBResetAllAutoSel.HMI2AllHMIAutoSel) OR ((#H_ActiveHMI = 3) AND #I_PBSetPBResetAllAutoSel.HMI3AllHMIAutoSel) OR ((#H_ActiveHMI = 4) AND #I_PBSetPBResetAllAutoSel.HMI4AllHMIAutoSel) OR ((#H_ActiveHMI = 5) AND #I_PBSetPBResetAllAutoSel.HMI5AllHMIAutoSel)) AND #ManualModeSel) OR ((#I_PBSetPBResetAllAutoSel.HMI1AllHMIAutoSel OR #I_PBSetPBResetAllAutoSel.HMI2AllHMIAutoSel OR #I_PBSetPBResetAllAutoSel.HMI3AllHMIAutoSel OR #I_PBSetPBResetAllAutoSel.HMI4AllHMIAutoSel OR #I_PBSetPBResetAllAutoSel.HMI5AllHMIAutoSel) AND NOT #ManualModeSel);
END_REGION

REGION Network 25: **** 5.2 - Equations - Flow **** Check Active HMI again - HMI <> 0
   // Check Active HMI again
   #CheckActiveHMI_2(IN := #H_ActiveHMI <> 0, PT := T#1s500ms);   // TON
   #CheckActiveHMI(IN := #CheckActiveHMI_2.Q, PT := T#1s500ms);   // TP
END_REGION

REGION Network 26: **** 5.2 - Equations - Flow **** Check Active HMI again - HMI = 0
   // Check Active HMI again
   #CheckActiveHMI_3(IN := #H_ActiveHMI = 0, PT := T#1s500ms);   // TON
   #CheckActiveHMI_1(IN := #CheckActiveHMI_3.Q, PT := T#1s500ms);   // TP
END_REGION

REGION Network 27: **** 7.3 - Submodules - Machine **** Process value
   // Process value
   #PV_PID := #PV_AIScaled;
END_REGION

REGION Network 28: **** 7.3 - Submodules - Machine **** Pid Controller
   // Pid Controller
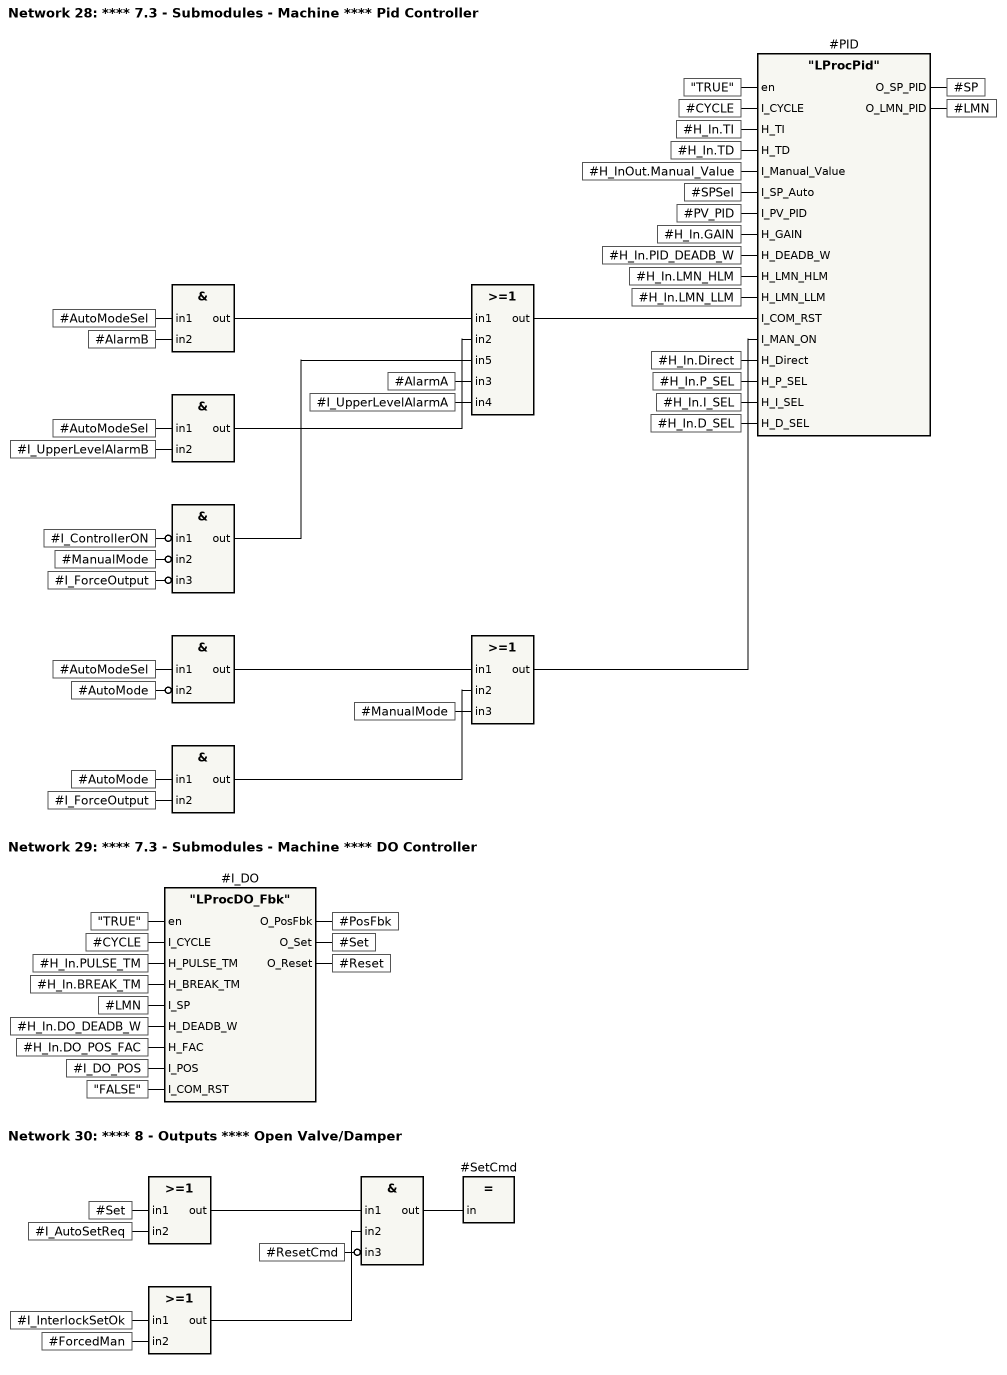
   IF "TRUE" THEN
       #PID(I_CYCLE := #CYCLE,   // "LProcPid"
            H_TI := #H_In.TI,
            H_TD := #H_In.TD,
            I_Manual_Value := #H_InOut.Manual_Value,
            I_SP_Auto := #SPSel,
            I_PV_PID := #PV_PID,
            H_GAIN := #H_In.GAIN,
            H_DEADB_W := #H_In.PID_DEADB_W,
            H_LMN_HLM := #H_In.LMN_HLM,
            H_LMN_LLM := #H_In.LMN_LLM,
            I_COM_RST := (#AutoModeSel AND #AlarmB) OR (#AutoModeSel AND #I_UpperLevelAlarmB) OR (NOT #I_ControllerON AND NOT #ManualMode AND NOT #I_ForceOutput) OR #AlarmA OR #I_UpperLevelAlarmA,
            I_MAN_ON := (#AutoModeSel AND NOT #AutoMode) OR (#AutoMode AND #I_ForceOutput) OR #ManualMode,
            H_Direct := #H_In.Direct,
            H_P_SEL := #H_In.P_SEL,
            H_I_SEL := #H_In.I_SEL,
            H_D_SEL := #H_In.D_SEL,
            O_SP_PID => #SP,
            O_LMN_PID => #LMN);
   END_IF;
END_REGION

REGION Network 29: **** 7.3 - Submodules - Machine **** DO Controller
   // DO Controller
   IF "TRUE" THEN
       #I_DO(I_CYCLE := #CYCLE,   // "LProcDO_Fbk"
             H_PULSE_TM := #H_In.PULSE_TM,
             H_BREAK_TM := #H_In.BREAK_TM,
             I_SP := #LMN,
             H_DEADB_W := #H_In.DO_DEADB_W,
             H_FAC := #H_In.DO_POS_FAC,
             I_POS := #I_DO_POS,
             I_COM_RST := "FALSE",
             O_PosFbk => #PosFbk,
             O_Set => #Set,
             O_Reset => #Reset);
   END_IF;
END_REGION

REGION Network 30: **** 8 - Outputs **** Open Valve/Damper
   // Open Valve/Damper
   #SetCmd := (#Set OR #I_AutoSetReq) AND (#I_InterlockSetOk OR #ForcedMan) AND NOT #ResetCmd;
END_REGION

REGION Network 31: **** 8 - Outputs **** Open Valve/Damper
   // Open Valve/Damper
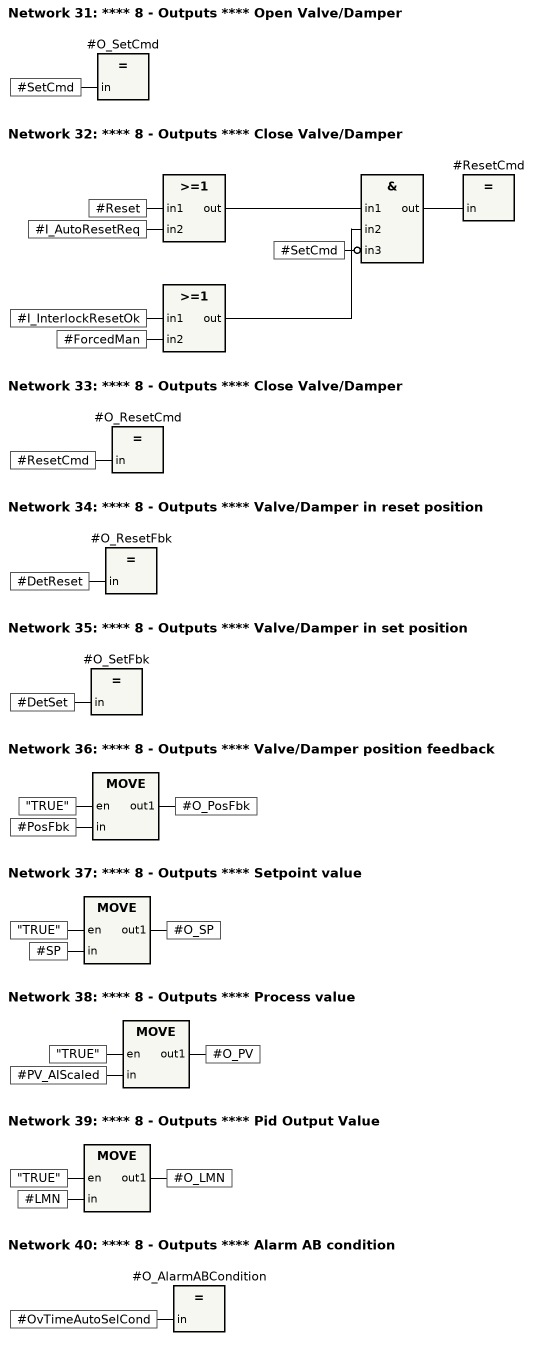
   #O_SetCmd := #SetCmd;
END_REGION

REGION Network 32: **** 8 - Outputs **** Close Valve/Damper
   // Close Valve/Damper
   #ResetCmd := (#Reset OR #I_AutoResetReq) AND (#I_InterlockResetOk OR #ForcedMan) AND NOT #SetCmd;
END_REGION

REGION Network 33: **** 8 - Outputs **** Close Valve/Damper
   // Close Valve/Damper
   #O_ResetCmd := #ResetCmd;
END_REGION

REGION Network 34: **** 8 - Outputs **** Valve/Damper in reset position
   // Valve/Damper in reset position
   #O_ResetFbk := #DetReset;
END_REGION

REGION Network 35: **** 8 - Outputs **** Valve/Damper in set position
   // Valve/Damper in set position
   #O_SetFbk := #DetSet;
END_REGION

REGION Network 36: **** 8 - Outputs **** Valve/Damper position feedback
   // Valve/Damper position feedback
   IF "TRUE" THEN #O_PosFbk := #PosFbk; END_IF;
END_REGION

REGION Network 37: **** 8 - Outputs **** Setpoint value
   // Setpoint value
   IF "TRUE" THEN #O_SP := #SP; END_IF;
END_REGION

REGION Network 38: **** 8 - Outputs **** Process value
   // Process value
   IF "TRUE" THEN #O_PV := #PV_AIScaled; END_IF;
END_REGION

REGION Network 39: **** 8 - Outputs **** Pid Output Value
   // Pid Output Value
   IF "TRUE" THEN #O_LMN := #LMN; END_IF;
END_REGION

REGION Network 40: **** 8 - Outputs **** Alarm AB condition
   // Alarm AB Condition
   #O_AlarmABCondition := #OvTimeAutoSelCond;
END_REGION

REGION Network 41: **** 9 - Alarm Summary **** Alarm A
   // Alarm A
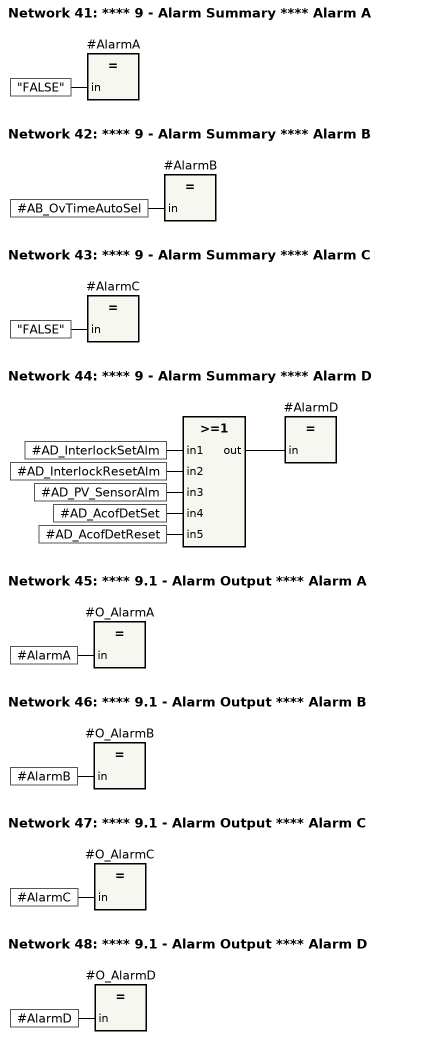
   #AlarmA := "FALSE";
END_REGION

REGION Network 42: **** 9 - Alarm Summary **** Alarm B
   // Alarm B
   #AlarmB := #AB_OvTimeAutoSel;
END_REGION

REGION Network 43: **** 9 - Alarm Summary **** Alarm C
   // Alarm C
   #AlarmC := "FALSE";
END_REGION

REGION Network 44: **** 9 - Alarm Summary **** Alarm D
   // Alarm D
   #AlarmD := #AD_InterlockSetAlm OR #AD_InterlockResetAlm OR #AD_PV_SensorAlm OR #AD_AcofDetSet OR #AD_AcofDetReset;
END_REGION

REGION Network 45: **** 9.1 - Alarm Output **** Alarm A
   // Alarm A
   #O_AlarmA := #AlarmA;
END_REGION

REGION Network 46: **** 9.1 - Alarm Output **** Alarm B
   // Alarm B
   #O_AlarmB := #AlarmB;
END_REGION

REGION Network 47: **** 9.1 - Alarm Output **** Alarm C
   // Alarm C
   #O_AlarmC := #AlarmC;
END_REGION

REGION Network 48: **** 9.1 - Alarm Output **** Alarm D
   // Alarm D
   #O_AlarmD := #AlarmD;
END_REGION

REGION Network 49: **** 9.2 - Alarm DWord**** Alarm To DWord
   // Alarm Word
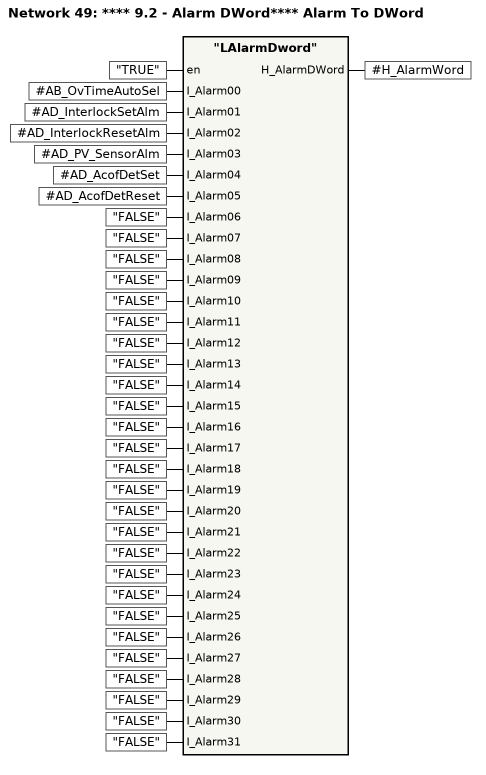
   IF "TRUE" THEN
       "LAlarmDword"(I_Alarm00 := #AB_OvTimeAutoSel,
                     I_Alarm01 := #AD_InterlockSetAlm,
                     I_Alarm02 := #AD_InterlockResetAlm,
                     I_Alarm03 := #AD_PV_SensorAlm,
                     I_Alarm04 := #AD_AcofDetSet,
                     I_Alarm05 := #AD_AcofDetReset,
                     I_Alarm06 := "FALSE",
                     I_Alarm07 := "FALSE",
                     I_Alarm08 := "FALSE",
                     I_Alarm09 := "FALSE",
                     I_Alarm10 := "FALSE",
                     I_Alarm11 := "FALSE",
                     I_Alarm12 := "FALSE",
                     I_Alarm13 := "FALSE",
                     I_Alarm14 := "FALSE",
                     I_Alarm15 := "FALSE",
                     I_Alarm16 := "FALSE",
                     I_Alarm17 := "FALSE",
                     I_Alarm18 := "FALSE",
                     I_Alarm19 := "FALSE",
                     I_Alarm20 := "FALSE",
                     I_Alarm21 := "FALSE",
                     I_Alarm22 := "FALSE",
                     I_Alarm23 := "FALSE",
                     I_Alarm24 := "FALSE",
                     I_Alarm25 := "FALSE",
                     I_Alarm26 := "FALSE",
                     I_Alarm27 := "FALSE",
                     I_Alarm28 := "FALSE",
                     I_Alarm29 := "FALSE",
                     I_Alarm30 := "FALSE",
                     I_Alarm31 := "FALSE",
                     H_AlarmDWord => #H_AlarmWord);
   END_IF;
END_REGION
END_FUNCTION_BLOCK
